// TIA Portal project "Lab01-git" (V16)

(* hardware
DEVICE "S7-1200 station_1"  S7-1200 Station
   slot 0: "Rack_0"  S7-1200 Rack  Rack  V1.0
   slot 1: "PLC_1"  CPU 1212C DC/DC/DC  6ES7 212-1AE40-0XB0  V4.4
*)

// ===== PLC "PLC_1"  CPU 1212C DC/DC/DC =====

VAR_GLOBAL   // PLC tag table "Tabla de variables estándar"
   "System_Byte" AT %MB1 : Byte;
   "FirstScan" AT %M1.0 : Bool;
   "DiagStatusUpdate" AT %M1.1 : Bool;
   "AlwaysTRUE" AT %M1.2 : Bool;
   "AlwaysFALSE" AT %M1.3 : Bool;
   "Clock_Byte" AT %MB0 : Byte;
   "Clock_10Hz" AT %M0.0 : Bool;
   "Clock_5Hz" AT %M0.1 : Bool;
   "Clock_2.5Hz" AT %M0.2 : Bool;
   "Clock_2Hz" AT %M0.3 : Bool;
   "Clock_1.25Hz" AT %M0.4 : Bool;
   "Clock_1Hz" AT %M0.5 : Bool;
   "Clock_0.625Hz" AT %M0.6 : Bool;
   "Clock_0.5Hz" AT %M0.7 : Bool;
   "input0_0" AT %I0.0 : Bool;
   "output0_0" AT %Q0.0 : Bool;
   "marca2_0" AT %M2.0 : Bool;
END_VAR

FUNCTION "FC_Clock" : Void   // FC1, LAD
{ S7_Optimized_Access := 'TRUE' }
VERSION : 0.1
   VAR_INPUT
      input : Bool;
      marca : Bool;
      clock : Bool;
   END_VAR
   VAR_OUTPUT
      output : Bool;
   END_VAR
BEGIN

REGION Network 1
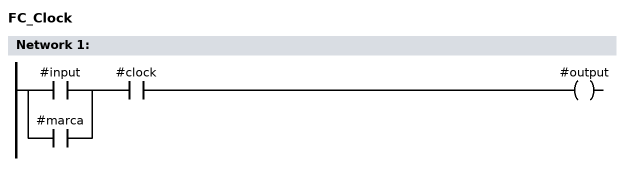
   RUNG wire#powerrail
      Contact( #input )
      wire#w1
      Contact( #clock )
      Coil( #output )
   END_RUNG
   RUNG wire#powerrail
      Contact( #marca )
   END_RUNG wire#w1
   // the same network as SCL:
   #output := (#input OR #marca) AND #clock;
END_REGION
END_FUNCTION

ORGANIZATION_BLOCK "Main"   // OB1, LAD, ProgramCycle
TITLE = "Main Program Sweep (Cycle)"
{ S7_Optimized_Access := 'TRUE' }
VERSION : 0.1
   VAR_INPUT
      Initial_Call : Bool;   // Initial call of this OB
      Remanence : Bool;   // =True, if remanent data are available
   END_VAR
BEGIN

REGION Network 1
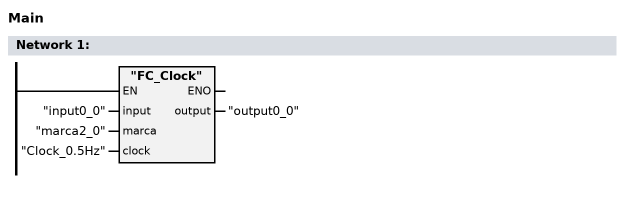
   RUNG wire#powerrail
      "FC_Clock"(input := "input0_0", marca := "marca2_0", clock := "Clock_0.5Hz", output => "output0_0")
   END_RUNG
   // the same network as SCL:
   "FC_Clock"(input := "input0_0", marca := "marca2_0", clock := "Clock_0.5Hz", output => "output0_0");
END_REGION
END_ORGANIZATION_BLOCK